{attribute 'qualified_only'}
VAR_GLOBAL
	MCP	: ST_Alarm_Base;
	Segment1 : ST_Alarm_Base;
	
	AlarmWord1  : ST_Alarm_Base;
	AlarmWord2  : ST_Alarm_Base;
	AlarmWord3  : ST_Alarm_Base;

END_VAR

(* stored: Version 1.1.0.1, ProductVersion 3.1.4024.11
   GVL Alarms_DB: Id {da78a859-3b87-44ba-a904-b3ed09d5c557} *)
